INTERFACE I_MutCTable EXTENDS I_CTable

METHOD Insert : Results.Result
VAR_INPUT
	iComponent	: I_Component;
END_VAR
VAR_OUTPUT
	nIndex		: UDINT;
END_VAR
END_METHOD

END_INTERFACE

(* stored: Version 1.1.0.1
   Itf I_MutCTable: Id {2cd7cdec-0286-4832-a950-30c990b9c773}
   Method Insert: Id {4c7ea171-4d2c-4d0a-84c7-27d6c43695f7} *)
